INTERFACE I_Mc3Axis_PTP EXTENDS I_Mc3Axis, I_AxisMoveAbsolute, I_AxisMoveModulo, I_AxisMoveRelative, I_AxisMoveVelocity

END_INTERFACE

(* stored: Version 1.1.0.1, ProductVersion 3.1.4026.20
   Itf I_Mc3Axis_PTP: Id {62de7262-895b-40fa-b1bf-5de4fead0c51} *)
